PROGRAM MAIN
VAR
	TONDelay: TON;
	TON_Delay: TON;
	TON_Timer: TON;
	blinkEnable: BOOL;
	TON_Blink1: TON;
	TON_Blink2: TON;
END_VAR

Blink();
Delay();
Timer();

ACTION Blink:
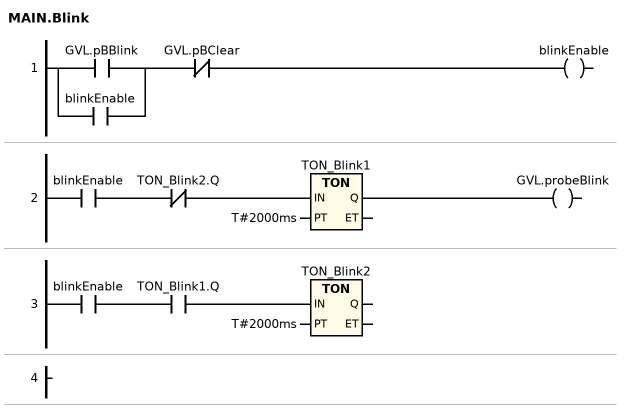
// NETWORK 1
blinkEnable := (GVL.pBBlink OR blinkEnable) AND NOT GVL.pBClear;

// NETWORK 2
TON_Blink1(IN := blinkEnable AND NOT TON_Blink2.Q, PT := T#2000ms); // TON
GVL.probeBlink := TON_Blink1.Q;

// NETWORK 3
TON_Blink2(IN := blinkEnable AND TON_Blink1.Q, PT := T#2000ms); // TON

// NETWORK 4
END_ACTION

ACTION Delay:
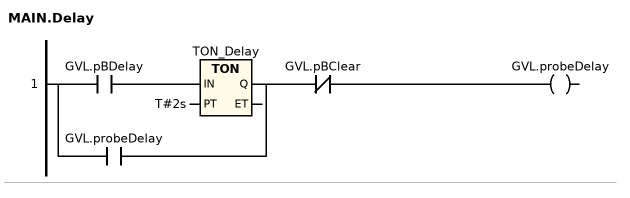
// NETWORK 1
TON_Delay(IN := GVL.pBDelay, PT := T#2s); // TON
GVL.probeDelay := (TON_Delay.Q OR GVL.probeDelay) AND NOT GVL.pBClear;
END_ACTION

ACTION Timer:
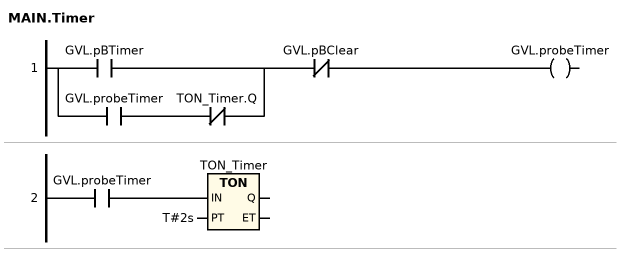
// NETWORK 1
GVL.probeTimer := (GVL.pBTimer OR GVL.probeTimer AND NOT TON_Timer.Q) AND NOT GVL.pBClear;

// NETWORK 2
TON_Timer(IN := GVL.probeTimer, PT := T#2s); // TON
END_ACTION

END_PROGRAM

(* stored: Version 1.1.0.1, ProductVersion 3.1.4024.12
   POU MAIN: Id {7571f8af-4de2-4e17-939f-a7e6f2a21ac7}, SpecialFunc None
   Action Blink: Id {b4a2e9d3-1af1-439b-b3e7-3b0c78cb338e}
   Action Delay: Id {b598e0f9-3e57-4f53-95b5-d572a60a8f4b}
   Action Timer: Id {a3a87c5a-5c45-4d05-ab1c-9e16233b5fb7} *)
